// TIA Portal V17 export
// export: Created 2022-02-03T14:45:13.1314747Z, ExportSetting WithDefaults, DisplayName Totally Integrated Automation Portal, DisplayVersion V17, DisplayName TIA Portal Openness, DisplayVersion V17, DisplayName TIA Portal Version Control Interface, DisplayVersion V17, DisplayName SINAMICS Startdrive Advanced, DisplayVersion V17, DisplayName SINAMICS Startdrive G130, G150, S120, S150, SINAMICS MV, S210, DisplayVersion V17, DisplayName SINAMICS Startdrive G110M, G120, G120C, G120D, G120P, G115D, DisplayVersion V17, DisplayName STEP 7 Professional, DisplayVersion V17, DisplayName STEP 7 Safety, DisplayVersion V17, DisplayName WinCC Advanced, DisplayVersion V17
FUNCTION "InitStore" : Void   // FC5, LAD
VERSION : 0.1
// stored: Access Published, AutoNumber true, IsIECCheckEnabled false, SetENOAutomatically false, UDAEnableTagReadback false
   VAR_INPUT
      all : Bool;
      currentStoreNo : UInt;
   END_VAR
   VAR_IN_OUT
      store : Array[0..9] of "typeStore";
   END_VAR
   VAR_TEMP
      tempCurrentStoreNo : UInt;
   END_VAR
BEGIN

REGION Network 1
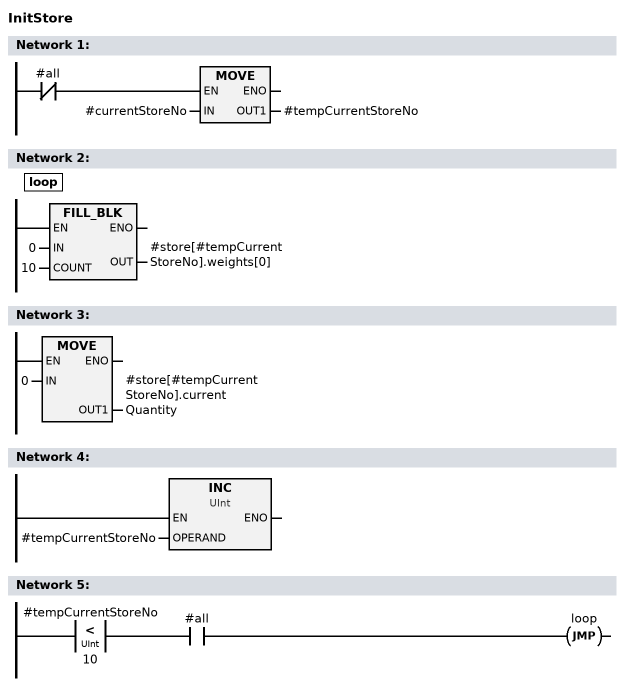
   RUNG wire#powerrail
      I_Contact( #all )
      Move(in := #currentStoreNo, out1 => #tempCurrentStoreNo)
   END_RUNG
   // the same network as SCL:
   IF NOT #all THEN #tempCurrentStoreNo := #currentStoreNo; END_IF;
END_REGION

REGION Network 2
   Label( loop )
   RUNG wire#powerrail
      FillBlockI(in := 0, count := 10, out => #store[#tempCurrentStoreNo].weights[0])
   END_RUNG
   // the same network as SCL:
   loop:
   FILL_BLK(IN := 0, COUNT := 10, OUT => #store[#tempCurrentStoreNo].weights[0]);
END_REGION

REGION Network 3
   RUNG wire#powerrail
      Move(in := 0, out1 => #store[#tempCurrentStoreNo].currentQuantity)
   END_RUNG
   // the same network as SCL:
   #store[#tempCurrentStoreNo].currentQuantity := 0;
END_REGION

REGION Network 4
   RUNG wire#powerrail
      { S7_Templates := "DestType := UInt" } Inc( #tempCurrentStoreNo )
   END_RUNG
   // the same network as SCL:
   #tempCurrentStoreNo := #tempCurrentStoreNo + 1;
END_REGION

REGION Network 5
   RUNG wire#powerrail
      { S7_Templates := "SrcType := UInt" } LT_Contact(in1 := #tempCurrentStoreNo, in2 := 10)
      Contact( #all )
      JumpCoil( loop )
   END_RUNG
   // the same network as SCL:
   IF (#tempCurrentStoreNo < 10) AND #all THEN GOTO loop; END_IF;
END_REGION
END_FUNCTION
